# EPICS substitutions: modules/event/evrSupport/Db/ioc/IOC-LI21-PM01pattern.substitutions
#
# Pattern records
file evrPatternAll.db {
#	    Device        ,  SLC Pattern, EVR/Trigger
#	                                    Links
  pattern { DEVICE        ,  LINK4      , LINK5 , LINK6 , TREF    , TS1ST, TS2ND }
	  { IOC:LI21:PM01 ,   ""        ,  ""   ,  ""   , 1.03E06 ,   1  ,   4   }
}
file evrEventAll.db {
  pattern { DEVICE        }
	  { IOC:LI21:PM01 }
}
